(* IEC 61131-3 sources: volt/packages/volt-lsp-iec/test-corpus/pro2193/Device/Plc Logic/Application/09 Misc/Library Manager/CmpVisuHandler, 42 files *)

(* ---- VISH_HAVETOMANAGECLIENT_DATA.dut ---- *)
TYPE VISH_HAVETOMANAGECLIENT_DATA :
STRUCT
	ISIZE : INT := SIZEOF(THIS^);
	DWEXTERNID : DWORD;
	DWFLAGS : DWORD;
END_STRUCT
END_TYPE

(* ---- VISH_HAVETOMANAGECLIENT_DATA2.dut ---- *)
TYPE VISH_HAVETOMANAGECLIENT_DATA2 :
STRUCT
	ISIZE : INT := SIZEOF(THIS^);
	DWEXTERNID : DWORD;
	DWFLAGS : DWORD;
	DWTAGSCAPACITY : DWORD;
	DWNUMTAGS : DWORD;
	PTAGS : POINTER TO Visu_ClientTagData;
END_STRUCT
END_TYPE

(* ---- VISH_HAVETOMANAGECLIENT_DATA3.dut ---- *)
TYPE VISH_HAVETOMANAGECLIENT_DATA3 :
STRUCT
	ISIZE : INT := SIZEOF(THIS^);
	DWEXTERNID : DWORD;
	DWFLAGS : DWORD;
	DWTAGSCAPACITY : DWORD;
	DWNUMTAGS : DWORD;
	PTAGS : POINTER TO Visu_ClientTagData;
	DWSESSIONID : DWORD;
END_STRUCT
END_TYPE

(* ---- VISH_STARTTARGETVISU_PARAMS.dut ---- *)
TYPE VISH_STARTTARGETVISU_PARAMS :
STRUCT
	ISIZE : INT := SIZEOF(THIS^);
	IXPOS : INT;
	IYPOS : INT;
	IWIDTH : INT;
	IHEIGHT : INT;
	STAPP : REFERENCE TO STRING;
END_STRUCT
END_TYPE

(* ---- VISH_STARTTARGETVISU_PARAMS2.dut ---- *)
TYPE VISH_STARTTARGETVISU_PARAMS2 :
STRUCT
	ISIZE : INT := SIZEOF(THIS^);
	IXPOS : INT;
	IYPOS : INT;
	IWIDTH : INT;
	IHEIGHT : INT;
	STAPP : REFERENCE TO STRING;
	UIANTIALIASING : UINT;
	UIWINDOWTYPE : UINT;
	UIUPDATERATEMS : UINT;
	UIFLAGS : UINT;
END_STRUCT
END_TYPE

(* ---- VISU_CLIENTTAGDATA.dut ---- *)
TYPE VISU_CLIENTTAGDATA :
STRUCT
	TAG : VisuEnumClientTag;
	STRVALUE : STRING(40);
END_STRUCT
END_TYPE

(* ---- VISU_INPUTCHECKS.dut ---- *)
TYPE VISU_INPUTCHECKS :
STRUCT
	IVERSION : INT := 1;
	PMIN : POINTER TO BYTE;
	PMAX : POINTER TO BYTE;
END_STRUCT
END_TYPE

(* ---- VISU_INPUTCHECKS2.dut ---- *)
TYPE VISU_INPUTCHECKS2 :
STRUCT
	IVERSION : INT := 2;
	PMIN : POINTER TO BYTE;
	PMAX : POINTER TO BYTE;
	DIMAXLEN : DINT;
END_STRUCT
END_TYPE

(* ---- VISU_TYPES.dut ---- *)
TYPE VISU_TYPES :
(
	TYPE_BOOL,
	TYPE_INT,
	TYPE_BYTE,
	TYPE_WORD,
	TYPE_DINT,
	TYPE_DWORD,
	TYPE_REAL,
	TYPE_TIME,
	TYPE_STRING,
	TYPE_ARRAY,
	TYPE_ENUM,
	TYPE_USERDEF,
	TYPE_BITORBYTE,
	TYPE_POINTER,
	TYPE_SINT,
	TYPE_USINT,
	TYPE_UINT,
	TYPE_UDINT,
	TYPE_DATE,
	TYPE_TOD,
	TYPE_DT,
	TYPE_VOID,
	TYPE_LREAL,
	TYPE_REF,
	TYPE_SUBRANGE,
	TYPE_LBITORBYTE,
	TYPE_LINT,
	TYPE_ULINT,
	TYPE_LWORD,
	TYPE_NONE,
	TYPE_BIT,
	TYPE_WSTRING,
	TYPE_LTIME,
	TYPE_LDATE,
	TYPE_LDT,
	TYPE_LTOD,
	MAXTYPES
);
END_TYPE

(* ---- VISUENUMCLIENTTAG.dut ---- *)
TYPE VISUENUMCLIENTTAG :
(
	UNDEFINED,
	NAME,
	ADDRESSIPV4
);
END_TYPE

(* ---- VISUSTRUCTEVENT.dut ---- *)
TYPE VISUSTRUCTEVENT :
STRUCT
	ISTRUCTSIZE : INT := SIZEOF(THIS^);
	EVENTTAG : DWORD := VISU_ET_MONITORING;
	DWPARAM1 : DWORD := 0;
	DWPARAM2 : DWORD := 0;
	CLIENTID : DWORD := 16#FFFFFFFF;
	DWADDDATASIZE : DWORD := 0;
	PADDITIONALDATA : POINTER TO BYTE;
	BIMPORTANTINPUT : BOOL;
	ROPTINVALIDRECT : VisuStructSimpleRectangle;
END_STRUCT
END_TYPE

(* ---- VISUSTRUCTEVENT2.dut ---- *)
TYPE VISUSTRUCTEVENT2 :
STRUCT
	LWIDSTACK : LWORD;
END_STRUCT
END_TYPE

(* ---- VISUSTRUCTPOINT.dut ---- *)
TYPE VISUSTRUCTPOINT :
STRUCT
	IX : INT;
	IY : INT;
END_STRUCT
END_TYPE

(* ---- VISUSTRUCTSIMPLERECTANGLE.dut ---- *)
TYPE VISUSTRUCTSIMPLERECTANGLE :
STRUCT
	PTTOPLEFT : VisuStructPoint;
	PTBOTTOMRIGHT : VisuStructPoint;
END_STRUCT
END_TYPE

(* ---- WEBSERVERINITPARAMETER.dut ---- *)
TYPE WEBSERVERINITPARAMETER :
STRUCT
	STSTARTHTMNAME : STRING;
END_STRUCT
END_TYPE

(* ---- CONSTANTS.gvl ---- *)
VAR_GLOBAL
	VISU_CLIENTS_NOTHINGTODO : INT := 16#0;
	VISU_CLIENTS_TOREMOVE : INT := 16#1;
	VISU_CLIENTS_TOADD : INT := 16#2;
	VISU_CLIENTS_INVALIDAPPLICATION : INT := 16#100;
	VISU_CLIENTS_CREATESHAREDMEMORY : DWORD := 16#1;
	VISU_CLIENTS_CREATEIECMEMORY : DWORD := 16#2;
	VISU_CLIENTS_PROGRAMMINGSYSTEM_OLD : DWORD := 16#10000;
	VISU_CLIENTS_STANDALONEVISU : DWORD := 16#20000;
	VISU_CLIENTS_HMI_TARGET : DWORD := 16#20000;
	VISU_CLIENTS_TARGETVISUALIZATION : DWORD := 16#40000;
	VISU_CLIENTS_WEBVISUALIZATION : DWORD := 16#80000;
	VISU_CLIENTS_PROGRAMMINGSYSTEM : DWORD := 16#200000;
	VISU_CLIENT_REMOVE : DWORD := 16#FFFFFFFE;
	VISU_STARTVISU_TARGETVISU : DWORD := 16#1;
	VISU_STARTVISU_WEBSERVER : DWORD := 16#2;
	VISU_STARTVISU_TARGETVISU_WITHRESULT : DWORD := 16#3;
	VISU_STARTVISU_TARGETVISU_CLOSE : DWORD := 16#4;
	VISU_STARTVISU_TARGETVISU_WITHRESULT2 : DWORD := 16#5;
	VISU_STARTVISU_WEBSERVER_RELEASE : DWORD := 16#6;
	VISU_STARTVISU_WEBSERVER_INITPARAMS : DWORD := 16#7;
	VISU_FCE_RESULT_OK : INT := 0;
	VISU_FCE_RESULT_PARAMETER : INT := 2;
	VISU_ET_NOTHING : DWORD := 16#0;
	VISU_ET_MONITORING : DWORD := 16#1;
	VISU_ET_MOUSEDOWN : DWORD := 16#2;
	VISU_ET_MOUSEUP : DWORD := 16#4;
	VISU_ET_MOUSEDBLCLK : DWORD := 16#8;
	VISU_ET_MOUSEMOVE : DWORD := 16#10;
	VISU_ET_MOUSEWHEEL : DWORD := 16#20;
	VISU_ET_INTERN_MOUSEOWNERSHIP : DWORD := 16#40;
	VISU_ET_KEYDOWN : DWORD := 16#80;
	VISU_ET_KEYUP : DWORD := 16#100;
	VISU_ET_CHAR : DWORD := 16#101;
	VISU_ET_EDITBOXRESULT : DWORD := 16#200;
	VISU_ET_INVALIDATETOOLTIP : DWORD := 16#201;
	VISU_ET_FILEDLGRESULT : DWORD := 16#202;
	VISU_ET_CALLNATIVECONTROLMETHODRESULT : DWORD := 16#203;
	VISU_ET_SETCLIENTSIZE : DWORD := 16#204;
	VISU_ET_CLIENTREQUEST : DWORD := 16#205;
	VISU_ET_MEASURESTRINGRESULT : DWORD := 16#206;
	VISU_ET_MEASURESTRING2RESULT : DWORD := 16#207;
	VISU_ET_ONDIALOGCLOSED : DWORD := 16#208;
	VISU_ET_PRINT : DWORD := 16#400;
	VISU_ET_GESTURE_EVENT_FLAG : DWORD := 16#800;
	VISU_ET_GESTURE_SPREADPINCH : DWORD := 16#801;
	VISU_ET_GESTURE_PAN : DWORD := 16#802;
	VISU_ET_GESTURE_FLICK : DWORD := 16#803;
	VISU_ET_GESTURE_IECTOUCH : DWORD := 16#804;
	VISU_ET_GESTURE_IECTOUCH_ONLYMOVES : DWORD := 16#805;
	VISU_ET_GESTURE_TOUCHTOMOUSE : DWORD := 16#806;
	VISU_ET_GESTURE_TOUCHTOMOUSE_ONLYMOVES : DWORD := 16#807;
	VISU_ET_MOUSEOUT : DWORD := 16#1000;
	VISU_ET_TOUCHSTART : DWORD := 16#1001;
	VISU_ET_TOUCHSTOP : DWORD := 16#1002;
	VISU_ET_INVALIDATE : DWORD := 16#100000;
	VISU_ET_SPECIAL : DWORD := 16#200000;
	VISU_ET_GENERAL : DWORD := 16#300000;
	VISU_GENTAG_REDUND_TICKET : DWORD := 16#1;
	VISU_INVTAG_SETSTARTVISU : DWORD := 16#1;
	VISU_INVTAG_SETSTARTVISU_NOTINITPAGE : DWORD := 16#2;
	VISU_INVTAG_EXTENSIBLE_FLAG : DWORD := 16#10000;
	VISU_INVTAG_EXTENSIBLE_CLIENTPAINTVER_FLAG : DWORD := 16#20000;
	VISU_INVTAG_EXTENSIBLE_CLIENTFEATURES_FLAG : DWORD := 16#40000;
	VISU_CLIENTVERSION_SUPPORTSEXTENDEDDRAWBUTTON : DWORD := 1;
	VISU_CLIENTVERSION_SUPPORTSPASSWORDINPUT : DWORD := 2;
	VISU_CLIENTVERSION_CORRECTED_RECT_DIMENSION : DWORD := 3;
	VISU_CLIENTVERSION_SUPPORTSDRAWPIXEL : DWORD := 4;
	VISU_CLIENTVERSION_OPTIMIZEDPAINTCOMMANDS : DWORD := 5;
	VISU_CLIENTREQUEST_RESTARTTARGETVISUIFNOTRUNNING : DWORD := 1;
	VISU_CLIENTVERSION_REMOVEALLTARGETVISUCLIENTS : DWORD := 2;
	VISU_CLIENTREQUEST_INVALIDATEALLCIENTS : DWORD := 3;
	VISU_STARTTARGETVISU_FLAGS_REMOTE : WORD := 16#1;
	VISU_STARTTARGETVISU_FLAGS_REMOTE_BESTFIT : WORD := 16#2;
	VISU_STARTTARGETVISU_FLAGS_MEASURE_PAINTCOMMANDEXECUTION : WORD := 16#4;
	VISU_STARTTARGETVISU_FLAGS_MEASURE_MOUSEDOWNREACTION : WORD := 16#8;
	VISU_STARTTARGETVISU_FLAGS_MEASURE_PAINTINGTOSCREEN : WORD := 16#10;
	VISU_STARTTARGETVISU_FLAGS_ACTIVATE_TOUCHHANDLING : WORD := 16#20;
	VISU_STARTTARGETVISU_FLAGS_OVERLAY : WORD := 16#200;
	VISU_STARTTARGETVISU_FLAGS_TRANSPARENT_BACKGROUND : WORD := 16#400;
	VIS_CLIENT_REGISTRATION_SUCCESSFULLY : DWORD := 16#0;
	VIS_CLIENT_REGISTRATION_NOT_REGISTERED : DWORD := 16#FFFFFFFF;
	VIS_CLIENT_REGISTRATION_NOT_YET_REGISTERED : DWORD := 16#FFFFFFFE;
	VIS_CLIENT_REGISTRATION_UNKNOWN_EXTERN_ID : DWORD := 16#FFFFFFFD;
END_VAR

(* ---- VERSIONCONSTANTS.gvl ---- *)
VAR_GLOBAL
	_CMPVISUHANDLER_VERSION_LARGEROREQUAL_3_5_17_0_ : INT := 0;
END_VAR

(* ---- VISHASSIGNRTSBASEDUSERMANAGEMENT.pou ---- *)
FUNCTION VISHASSIGNRTSBASEDUSERMANAGEMENT : RTS_IEC_RESULT
VAR_INPUT
	XRTSBASEDACTIVE : BOOL;
	XRESET : BOOL;
END_VAR
END_FUNCTION

(* ---- VISHBUFFERPRINTF.pou ---- *)
FUNCTION VISHBUFFERPRINTF : INT
VAR_INPUT
	PSTFORMAT : POINTER TO STRING;
	PVARADR : POINTER TO DWORD;
	DWVARTYPE : DWORD;
	PBUFFER : POINTER TO BYTE;
	DWBUFFERSIZE : UDINT;
END_VAR
END_FUNCTION

(* ---- VISHBUFFERPRINTFW.pou ---- *)
FUNCTION VISHBUFFERPRINTFW : INT
VAR_INPUT
	WSTFORMAT : POINTER TO WSTRING;
	PVARADR : POINTER TO DWORD;
	DWVARTYPE : DWORD;
	PBUFFER : POINTER TO BYTE;
	DWBUFFERSIZE : UDINT;
END_VAR
END_FUNCTION

(* ---- VISHCLIENTCREATE.pou ---- *)
FUNCTION VISHCLIENTCREATE : INT
VAR_INPUT
	STAPPNAME : STRING;
	CLIENTTYPE : UINT;
	DWEXTERNID : DWORD;
	DWCREATIONFLAGS : DWORD;
	NUMTAGS : INT;
	PTAGS : POINTER TO Visu_ClientTagData;
END_VAR
VAR_OUTPUT
	DWEXTERNIDCREATED : DWORD;
END_VAR
END_FUNCTION

(* ---- VISHCLIENTGETINFO.pou ---- *)
FUNCTION VISHCLIENTGETINFO : INT
VAR_INPUT
	DWEXTERNID : DWORD;
	PTAGS : POINTER TO Visu_ClientTagData;
	ISZTAGS : INT;
END_VAR
VAR_OUTPUT
	DWCREATIONFLAGS : DWORD;
	INUMTAGS : INT;
END_VAR
END_FUNCTION

(* ---- VISHCLIENTKEEPALIVE.pou ---- *)
FUNCTION VISHCLIENTKEEPALIVE
VAR_INPUT
	DWEXTERNID : DWORD;
END_VAR
END_FUNCTION

(* ---- VISHCLIENTREMOVE.pou ---- *)
FUNCTION VISHCLIENTREMOVE : INT
VAR_INPUT
	DWEXTERNID : DWORD;
END_VAR
END_FUNCTION

(* ---- VISHCONFIGUREEVENTBUFFER.pou ---- *)
FUNCTION VISHCONFIGUREEVENTBUFFER : RTS_IEC_RESULT
VAR_INPUT
	STAPPNAME : STRING;
	BUFFERSIZE : UINT;
	EVENTEXTENSIONSIZE : UINT;
	XMERGEEVENTS : BOOL;
END_VAR
END_FUNCTION

(* ---- VISHFILLCURRENTEVENT.pou ---- *)
FUNCTION VISHFILLCURRENTEVENT : INT
VAR_INPUT
	STAPPNAME : STRING;
	PEVENT : POINTER TO VisuStructEvent;
END_VAR
END_FUNCTION

(* ---- VISHGETCLIENTID.pou ---- *)
FUNCTION VISHGETCLIENTID : INT
VAR_INPUT
	DWEXTERNID : DWORD;
END_VAR
END_FUNCTION

(* ---- VISHGETCURRENTEVENT.pou ---- *)
FUNCTION VISHGETCURRENTEVENT : VisuStructEvent
VAR_INPUT
	STAPPNAME : STRING;
END_VAR
END_FUNCTION

(* ---- VISHGETCURRENTEVENT2.pou ---- *)
FUNCTION VISHGETCURRENTEVENT2 : POINTER TO VisuStructEvent2
VAR_IN_OUT
	STAPPNAME : STRING;
END_VAR
END_FUNCTION

(* ---- VISHHAVETOMANAGECLIENTS.pou ---- *)
FUNCTION VISHHAVETOMANAGECLIENTS : INT
VAR_INPUT
	PDATA : REFERENCE TO Vish_HavetomanageClient_Data;
	STAPPNAME : STRING;
END_VAR
END_FUNCTION

(* ---- VISHHAVETOMANAGECLIENTS2.pou ---- *)
FUNCTION VISHHAVETOMANAGECLIENTS2 : INT
VAR_INPUT
	PDATA : POINTER TO Vish_HavetomanageClient_Data2;
	STAPPNAME : STRING;
END_VAR
END_FUNCTION

(* ---- VISHHAVETOMANAGECLIENTS3.pou ---- *)
FUNCTION VISHHAVETOMANAGECLIENTS3 : INT
VAR_INPUT
	PDATA : POINTER TO Vish_HavetomanageClient_Data3;
	STAPPNAME : STRING;
END_VAR
END_FUNCTION

(* ---- VISHISCLIENTREGISTERED.pou ---- *)
FUNCTION VISHISCLIENTREGISTERED : DWORD
VAR_INPUT
	DWEXTERNID : DWORD;
END_VAR
END_FUNCTION

(* ---- VISHLOCKCLIENTCREATION.pou ---- *)
FUNCTION VISHLOCKCLIENTCREATION : INT
VAR_INPUT
	STAPPNAME : STRING;
	DWTYPE : DWORD;
END_VAR
VAR_OUTPUT
	ILOCKCOUNT : INT;
END_VAR
END_FUNCTION

(* ---- VISHPRINTF.pou ---- *)
FUNCTION VISHPRINTF : POINTER TO STRING
VAR_INPUT
	PSTFORMAT : POINTER TO STRING;
	PVARADR : POINTER TO DWORD;
	DWVARTYPE : DWORD;
END_VAR
END_FUNCTION

(* ---- VISHPRINTFW.pou ---- *)
FUNCTION VISHPRINTFW : POINTER TO WSTRING
VAR_INPUT
	PWSTFORMAT : POINTER TO WSTRING;
	PVARADR : POINTER TO DWORD;
	DWVARTYPE : DWORD;
END_VAR
END_FUNCTION

(* ---- VISHREMOVEALLCLIENT.pou ---- *)
FUNCTION VISHREMOVEALLCLIENT : INT
VAR_INPUT
	STAPPNAME : STRING;
	DWTYPE : DWORD;
END_VAR
VAR_OUTPUT
	ICNTREMOVED : INT;
END_VAR
END_FUNCTION

(* ---- VISHREMOVECURRENTEVENT.pou ---- *)
FUNCTION VISHREMOVECURRENTEVENT : INT
VAR_INPUT
	STAPPNAME : STRING;
END_VAR
END_FUNCTION

(* ---- VISHSETCLIENTDATA.pou ---- *)
FUNCTION VISHSETCLIENTDATA : INT
VAR_INPUT
	DWEXTERNID : DWORD;
	ICLIENTID : INT;
	PPAINTBUFFER : POINTER TO BYTE;
	STAPPNAME : STRING;
END_VAR
END_FUNCTION

(* ---- VISHSTARTVISU.pou ---- *)
FUNCTION VISHSTARTVISU : INT
VAR_INPUT
	DWTYPE : DWORD;
	DWPARAM1 : __XWORD;
	DWPARAM2 : __XWORD;
END_VAR
END_FUNCTION

(* ---- VISHUNLOCKCLIENTCREATION.pou ---- *)
FUNCTION VISHUNLOCKCLIENTCREATION : INT
VAR_INPUT
	STAPPNAME : STRING;
END_VAR
VAR_OUTPUT
	ILOCKCOUNT : INT;
END_VAR
END_FUNCTION

(* ---- VISHWRITEVALUEIFVALID.pou ---- *)
FUNCTION VISHWRITEVALUEIFVALID : INT
VAR_INPUT
	PSTTOWRITE : POINTER TO STRING;
	PDATATOWRITETO : POINTER TO BYTE;
	DATATYPE : Visu_Types;
	PINPUTCHECKS : POINTER TO Visu_InputChecks;
END_VAR
END_FUNCTION
